// TIA Portal V20 export
DATA_BLOCK "BK27"   // DB255
// stored: MemoryReserve 100
   VAR
      "X10-1.SPARE" : Bool := FALSE;
      "X11-1.JR WINDER CLAMP BTM REAR UP/DOWN" : Bool := FALSE;
      "X12-1.SPARE" : Bool := FALSE;
      "X13-1.JR WINDER CLAMP BTM FRONT UP/DOWN" : Bool := FALSE;
      "X14-1.SPARE" : Bool := FALSE;
      "X15-1.JR WINDER CLAMP FRONT TOP PRESSURE SWITCH" : Bool := FALSE;
      "X16-1.JR WINDER STACK DETECT SENSOR" : Bool := FALSE;
      "X17-1.SPARE" : Bool := FALSE;
      "X10-2.SPARE" : Bool := FALSE;
      "X11-2.SPARE" : Bool := FALSE;
      "X12-2.SPARE" : Bool := FALSE;
      "X13-2.SPARE" : Bool := FALSE;
      "X14-2.SPARE" : Bool := FALSE;
      "X15-2.JR WINDER CLAMP FRONT BTM PRESSURE SWITCH" : Bool := FALSE;
      "X16-2.SPARE" : Bool := FALSE;
      "X17-2.SPARE" : Bool := FALSE;
   END_VAR
BEGIN
END_DATA_BLOCK
